# EPICS substitutions: iocBoot/ioc13PECell/asynRecord.substitutions
file "$(ASYN)/db/asynRecord.db"
{
pattern
{P           R         PORT    ADDR    OMAX  IMAX}
{13PECELL:  asyn_1   serial1    0     256  256}
{13PECELL:  asyn_2   serial2    0     256  256}
}
